PROGRAM MAIN
VAR		
	bRun	:	BOOL := FALSE;
	
	secondtimer	:	TimerCounter;
	
	oversamplingHandler	:	OversamplingHandler;
	
	//EL3751 signals in
	voltageIn	AT%I*	:	DINT;
	voltageIn2	AT%I*	:	DINT;
	
	EL3xxx	:	AnalogSignalProcessing;
	ELM3xxx	:	AnalogSignalProcessing;
	
	primaryVoltage		: LREAL;
	secondaryVoltage	:	LREAL;
	
	//scope server control block
(*	fbScopeServer	:	FB_ScopeServerSample;
	xStartStopScope	:	BOOL;
	*)
	
	//Analytics Teach FB
	//fbTimeTeach	:	TimeBasedTeach;
	
	// dc time stuff
	fbSystemDCTime	:	GetDCTime;
END_VAR

IF bRun THEN
		
	//Timer counter fb
	//secondtimer();
	
	//oversampling - ELM3002 processing
	oversamplingHandler();
	
	//EL3751 reading signal
	(*EL3xxx(signalIn := voltageIn);
	ELM3xxx(signalIn := voltageIn2);*)
	
	//EL3751 Signal processing
	//primaryVoltage := EL3xxx.voltageIn;
	//secondaryVoltage := ELM3xxx.voltageIn;
	
	//Scope server control from PLC
	(*
	fbScopeServer(
		sNetId					:='5.119.159.52.1.1', 
		bExternalTriggerEvent	:=xStartStopScope , 
		sConfigFile				:= 'C:\Y.tcscopex', 
		sSaveFile				:='C:\Record.svdx' , 
		bBusy					=> , 
		bError					=>, 
		nErrorId				=>);
	*)
	
	//fbTimeTeach();

	fbSystemDCTime();
	
END_IF

bRun := True;

END_PROGRAM

(* stored: Version 1.1.0.1, ProductVersion 3.1.4024.12
   POU MAIN: Id {e6967ea9-cb30-4ee7-b42c-ad0177bcac3f}, SpecialFunc None *)
